{attribute 'qualified_only'}
{attribute 'strict'}
TYPE E_JogFrame :
(
    Base   := 0,
    Tool   := 1,
    Custom := 2
);
END_TYPE

(* stored: Version 1.1.0.1, ProductVersion 3.1.4026.18
   DUT E_JogFrame: Id {026c7766-cf73-4abf-954f-d3ce0f07ac09} *)
